FUNCTION PositionF_CurrentCoeff : LREAL
VAR_INPUT
    Current : LREAL;
END_VAR
VAR
END_VAR

PositionF_CurrentCoeff   := (-0.0009*Current)+ 1.0016;

END_FUNCTION

(* stored: Version 1.1.0.1
   POU PositionF_CurrentCoeff: Id {dd4ad5d7-76cc-0a09-00fd-b2e01a0ea7b8}, SpecialFunc None *)
